Fanuc KAREL source: kf00111.KL

-- PROVISIONAL review KL for V770-1; original PC SHA256 513b5e278a55b578d3d80cf76ced12d39a655bd52130387341b3e0fac50d49fe
-- Incomplete behavior may be omitted. Consult companion uncertainty JSON. Do not deploy.
PROGRAM KF00111
%NOLOCKGROUP
VAR
  I : INTEGER
  J : INTEGER
  X : REAL
  Y : REAL
  B : BOOLEAN
  C : BOOLEAN
  TXT : STRING[80]
  TXT2 : STRING[80]
  STATUS : INTEGER
-- UNRESOLVED_DECL AI type=002010
-- UNRESOLVED_DECL BI type=002010
-- UNRESOLVED_DECL P type=000102
-- UNRESOLVED_DECL JP type=000199
-- UNRESOLVED_DECL PF type=000101
-- UNRESOLVED_DECL V1 type=000013
-- UNRESOLVED_DECL V2 type=000013
BEGIN
  -- UNRESOLVED_PC offsets 5-12; opcodes 9D,23
  -- UNRESOLVED_PC offsets 17-28; opcodes 2E,23
  -- UNRESOLVED_PC offsets 33-40; opcodes 9D,23
  -- UNRESOLVED_PC offsets 45-55; opcodes 9D,19,64,23
  -- UNRESOLVED_PC offsets 60-64; opcodes 7F
END KF00111
